ABB RobotStudio station: IRB120_RBE502_Station.rsstn

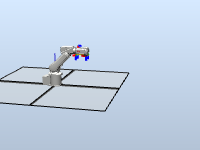
Station IRB120_RBE502_Station (saved by RobotStudio 6.8.8307.1040)
Controller RBE502_Proj
  mechanical unit ROB_1: IRB120_3_58__01, 6 joints, base frame (0, 0, 0) mm
Layout (positions relative to the parent item):
  - IRB120_3_58__01 [mechanism, from Robots\IRB120_3_58_G_01.rslib] at (0, 0, 0) mm; joint values [0, 0.7809, -0.7816, 0, 1.5715, 0] (rad or m)
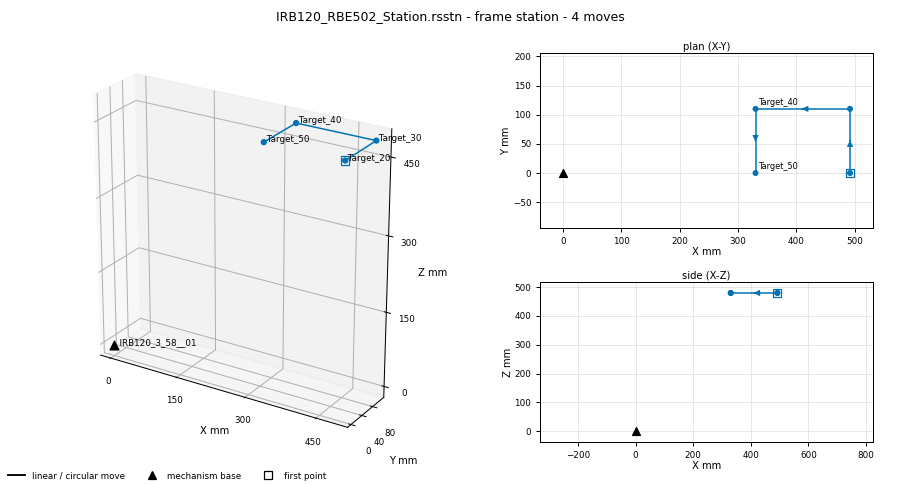
[picture p0: tool path of IRB120_RBE502_Station.rsstn in frame station, 4 of 6 moves have a stored position in this frame; points joined in program order, loops and branches not executed]
Targets, tools, work objects and paths stored in the station, written as RAPID:
! task T_ROB1
MODULE CalibData
  TASK PERS wobjdata RBE502_SqTest:=[FALSE,TRUE,"",[[0,0,0],[1,0,0,0]],[[0,0,0],[1,0,0,0]]];
  TASK PERS tooldata tool1:=[TRUE,[[0,0,0],[1,0,0,0]],[1,[0,0,1],[1,0,0,0],0,0,0]];
ENDMODULE

! task T_ROB1
MODULE Module1
  CONST robtarget Target_10:=[[448.631061346,0,135.404128273],[0.010002859,0,0.99994997,0],[0,0,0,0],[9E+09,9E+09,9E+09,9E+09,9E+09,9E+09]];
  CONST robtarget Target_20:=[[492,0,480],[0.010002835,0.00000001,0.99994997,-0.00000001],[0,-1,0,0],[9E+09,9E+09,9E+09,9E+09,9E+09,9E+09]];
  CONST robtarget Target_30:=[[492,110,480],[0.010002818,0.000000017,0.999949971,-0.000000017],[0,-1,0,0],[9E+09,9E+09,9E+09,9E+09,9E+09,9E+09]];
  CONST robtarget Target_40:=[[330,110,480],[0.010002809,0.000000017,0.999949971,-0.000000017],[0,-1,0,0],[9E+09,9E+09,9E+09,9E+09,9E+09,9E+09]];
  CONST robtarget Target_50:=[[330,0,480],[0.010002809,0.000000017,0.999949971,-0.000000017],[0,-1,0,0],[9E+09,9E+09,9E+09,9E+09,9E+09,9E+09]];
  PROC Path_Sq()
    MoveL Target_20,v500,z10,tool0\WObj:=RBE502_SqTest;
    MoveL Target_30,v500,z10,tool0\WObj:=RBE502_SqTest;
    MoveL Target_40,v500,z10,tool0\WObj:=RBE502_SqTest;
    MoveL Target_50,v500,z10,tool0\WObj:=RBE502_SqTest;
  ENDPROC
  PROC main()
    MoveAngleMatlab;
  ENDPROC
ENDMODULE

! task T_ROB1
MODULE Test_MoveAbsJ
  VAR jointtarget rotJoints:=[[0,0,0,0,0,0],[9E+09,9E+09,9E+09,9E+09,9E+09,9E+09]];
  PROC MoveAbsJ_test()
    MoveAbsJ rotJoints,v500,z10,tool0\WObj:=RBE502_SqTest;
  ENDPROC
  PROC MoveAngleMatlab()
    MoveAbsJ rotJoints,v500,z10,tool0\WObj:=RBE502_SqTest;
  ENDPROC
ENDMODULE

